# EPICS substitutions: example/exampleApp/Db/example.substitutions
file tdklambda.template
{
  pattern {   name,          ps,   grp  , drvl,  drvh, vdrvh }
          {bl99:tdklambda,    ps1,  Dipole,  0  ,  5  ,  12  }
}
